{attribute addProperty BoxType "EL6002-0000-0019"}
{attribute addProperty Id "CtrlAT %Q*Ctrl_4B42712A5Data_OutAT %Q*ARRAY[0..21] OF USINT22"}
{attribute addProperty CRC "3056402346"}
{attribute addProperty SizeInBites "216"}
{attribute addProperty SizeInBytes "27"}
TYPE COM_RxPDO_Map_Outputs_Channel_476040AE :
STRUCT
	{attribute addProperty Name "Ctrl"}
	Ctrl AT %Q* : Ctrl_4B42712A;
	{attribute addProperty Name "Data_Out"}
	Data_Out AT %Q* : ARRAY[0..21] OF USINT;
END_STRUCT
END_TYPE

(* stored: Version 1.2.0.0, ProductVersion 3.1.4024.9
   DUT COM_RxPDO_Map_Outputs_Channel_476040AE: Id {5517d9f4-f2d3-4c00-b856-3fe932b240f1} *)
